Yaskawa INFORM job: REF_ODWLOK_NEW_X2.JBI

/JOB
//NAME REF_ODWLOK_NEW_X2
///FOLDERNAME INNE
//POS
///NPOS 13,13,0,0,0,0
///TOOL 0
///POSTYPE PULSE
///PULSE
C00000=29141,230992,241019,-120436,-126056,-18240
C00001=-85879,-96353,-67507,26769,-8866,29155
C00002=-90682,-94952,-60903,2018,-11322,40048
C00003=-108098,-110399,-80759,-62152,-14175,68196
C00004=-113513,-107421,-73683,-61030,-18975,67386
C00005=-144153,-52243,-78334,-12318,21797,-35843
C00006=-101212,-47573,-19223,-109162,37686,9551
C00007=221370,-128165,-94668,86127,-52368,4397
C00008=222637,-115629,-85020,86703,-53233,4058
C00009=226166,-95549,-92179,97275,-55828,-4226
C00010=227012,-86748,-82897,96365,-56343,-3549
C00011=228844,-77551,-114266,109939,-62245,-16021
C00012=231303,-85254,-61893,88675,-59409,3048
BC00000=270176,1327400,971
BC00001=7,705730,699321
BC00002=7,705730,699321
BC00003=7,705730,699321
BC00004=7,705730,699321
BC00005=69542,664684,1004097
BC00006=69542,664684,1004095
BC00007=188146,1353181,597486
BC00008=188146,1353181,597486
BC00009=188146,1353181,597486
BC00010=188146,1353181,597486
BC00011=208965,1347150,856546
BC00012=208965,1347150,856546
//INST
///DATE 2024/02/01 20:12
///ATTR SC,RW
///GROUP1 RB1,BS1
NOP
'FRONT
MOVJ C00000 BC00000 VJ=0.78 PL=0  //FRONT_RIGHT
'LEFT
COMM MOVJ C00001 BC00001 VJ=0.78 PL=0  //1_SMALL
COMM MOVJ C00002 BC00002 VJ=0.78 PL=0  //2_SMALL
COMM MOVJ C00003 BC00003 VJ=0.78 PL=0  //3_SMALL
COMM MOVJ C00004 BC00004 VJ=0.78 PL=0  //4_SMALL
MOVJ C00005 BC00005 VJ=0.78 PL=0  //1_LARGE
MOVJ C00006 BC00006 VJ=0.78 PL=0  //2_SMALL
'RIGHT
COMM MOVJ C00007 BC00007 VJ=0.78 PL=0  //1_SMALL
COMM MOVJ C00008 BC00008 VJ=0.78 PL=0  //2_SMALL
COMM MOVJ C00009 BC00009 VJ=0.78 PL=0  //3_SMALL
COMM MOVJ C00010 BC00010 VJ=0.78 PL=0  //4_SMALL
MOVJ C00011 BC00011 VJ=0.78 PL=0  //1_LARGE
MOVJ C00012 BC00012 VJ=0.78 PL=0  //2_SMALL
END
